TYPE ST_EL2574_ExtendedMode :
	STRUCT
		In	AT %I* : ST_EL2574_In;
		Out AT %Q* : ST_EL2574_Out;
	END_STRUCT
END_TYPE

(* stored: Version 1.1.0.1
   DUT ST_EL2574_ExtendedMode: Id {437d2004-9336-408a-b214-9060ecc066dd} *)
